{attribute 'linkalways'} 
{attribute 'no_explicit_call' := 'This FB is a CLASS and must be accessed using methods or properties'}
{attribute 'enable_dynamic_creation'}
FUNCTION_BLOCK FINAL OR_LWORD EXTENDS Node
VAR
	in1 : _LWORD(0);
	in2 : _LWORD(0);
	out : _LWORD(0);
END_VAR

METHOD PUBLIC Clone : I_Node
VAR
	pNode : POINTER TO OR_LWORD;
END_VAR
pNode := __NEW(OR_LWORD);
Clone := pNode^;
END_METHOD

METHOD FB_init : BOOL
VAR_INPUT
	bInitRetains : BOOL; // if TRUE, the retain variables are initialized (warm start / cold start)
	bInCopyCode : BOOL;  // if TRUE, the instance afterwards gets moved into the copy code (online change)
END_VAR
AddInput('in1',THIS^.in1);
AddInput('in2',THIS^.in2);
AddOutput('out', THIS^.out);
END_METHOD

METHOD PROTECTED OnExecute
VAR
END_VAR
out.Value := in1.Value OR in2.Value;
END_METHOD

END_FUNCTION_BLOCK

(* stored: Version 1.1.0.1, ProductVersion 3.1.4024.15
   POU OR_LWORD: Id {cc719bbc-f061-4088-b85c-17f56ce486f3}, SpecialFunc None
   Folder Constructor: Id {8ef0fb75-5cfb-4d4c-a4d5-bb7d0f5f653f}
   Method Clone: Id {dfcff91c-1df2-40e4-a8d7-f552d3475af8}
   Method FB_init: Id {5964542b-3445-4f0a-bb91-907a39e2ba76}
   Method OnExecute: Id {c7f43228-08db-4b6c-bd90-7184d21f9476} *)
